FUNCTION_BLOCK FB_Carro_GRF_SFC
// Transcripción del grafcet (GRF -> SFC)
VAR_INPUT
    ManiobrasTotales: UINT := 2;
    TiempoEspera: TIME := T#2S;
END_VAR
VAR_OUTPUT
    ManiobrasPendientes: UINT;
    TiempoPendiente: TIME;
END_VAR
VAR
    // Bloques funcionales
    FlancoPulsadorMarcha: R_TRIG;
    Intermitencia: FB_Blink;
    
    // Entradas
    i_PulsadorMarcha AT %I*: BOOL;
    i_FinalCarreraIzquierda AT %I*: BOOL := TRUE;
    i_FinalCarreraDerecha AT %I*: BOOL;
    
    // Salidas
    o_MarchaIzquierda AT %I*: BOOL;
    o_MarchaDerecha AT %I*: BOOL;
    o_LamparaMarcha AT %I*: BOOL;
END_VAR

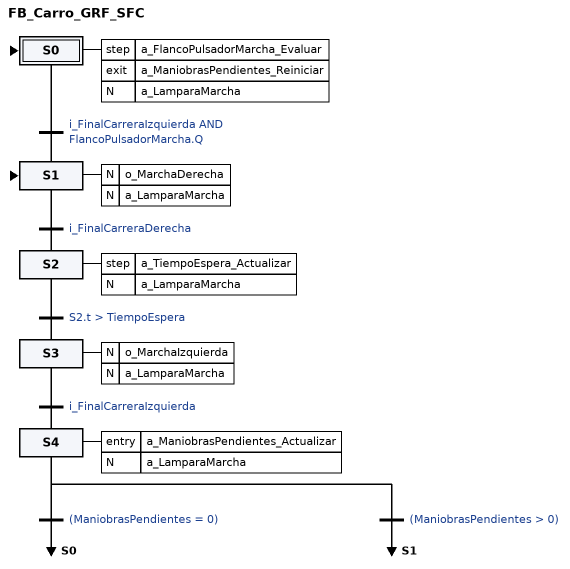
INITIAL_STEP S0:
    a_FlancoPulsadorMarcha_Evaluar(N);  // step action
    a_ManiobrasPendientes_Reiniciar(P0);  // exit action
    a_LamparaMarcha(N);
END_STEP
TRANSITION FROM S0 TO S1
    := i_FinalCarreraIzquierda AND FlancoPulsadorMarcha.Q;
END_TRANSITION
STEP S1:
    o_MarchaDerecha(N);
    a_LamparaMarcha(N);
END_STEP
TRANSITION FROM S1 TO S2
    := i_FinalCarreraDerecha;
END_TRANSITION
STEP S2:
    a_TiempoEspera_Actualizar(N);  // step action
    a_LamparaMarcha(N);
END_STEP
TRANSITION FROM S2 TO S3
    := S2.t > TiempoEspera;
END_TRANSITION
STEP S3:
    o_MarchaIzquierda(N);
    a_LamparaMarcha(N);
END_STEP
TRANSITION FROM S3 TO S4
    := i_FinalCarreraIzquierda;
END_TRANSITION
STEP S4:
    a_ManiobrasPendientes_Actualizar(P1);  // entry action
    a_LamparaMarcha(N);
END_STEP
TRANSITION FROM S4 TO S0
    := (ManiobrasPendientes = 0);
END_TRANSITION
TRANSITION FROM S4 TO S1
    := (ManiobrasPendientes > 0);
END_TRANSITION

ACTION a_FlancoPulsadorMarcha_Evaluar:
FlancoPulsadorMarcha(CLK := i_PulsadorMarcha);
END_ACTION

ACTION a_LamparaMarcha:
Intermitencia(Enable := S0.x);

o_LamparaMarcha := (S0.x AND Intermitencia.Q) OR S1.x OR S2.x OR S3.x OR S4.x;
END_ACTION

ACTION a_ManiobrasPendientes_Actualizar:
IF (ManiobrasPendientes > 0) THEN
    ManiobrasPendientes := ManiobrasPendientes - 1;
END_IF;
END_ACTION

ACTION a_ManiobrasPendientes_Reiniciar:
ManiobrasPendientes := ManiobrasTotales;
END_ACTION

ACTION a_TiempoEspera_Actualizar:
IF TiempoEspera >= S2.t THEN
    TiempoPendiente := TiempoEspera - S2.t;
END_IF;
END_ACTION

END_FUNCTION_BLOCK

(* stored: Version 1.1.0.1, ProductVersion 3.1.4024.16
   POU FB_Carro_GRF_SFC: Id {22d700f1-c096-431a-babb-bbf0219d1b28}, SpecialFunc None
   Action a_FlancoPulsadorMarcha_Evaluar: Id {270c1a7b-d542-42d7-8ec5-6ffc85e0e9de}
   Action a_LamparaMarcha: Id {6e036b04-25c8-412d-a86f-80391637dfaf}
   Action a_ManiobrasPendientes_Actualizar: Id {5d28dd82-84ca-4aee-a032-3a689682c7af}
   Action a_ManiobrasPendientes_Reiniciar: Id {c7170512-a360-4839-85df-b664689808ff}
   Action a_TiempoEspera_Actualizar: Id {e0af001b-8951-4d88-ba0a-a0414f07cb8b} *)
